# EPICS StreamDevice protocol: epics_installer_v1.0/option/serialTest_RAON_20220420/db/A100L.proto
ReplyTimeout = 500;
InTerminator = CR;

# No outTerminator because we need to send ENQ clean or RS485 will mess up the reply.

#address = ESC "0\$1"; # for RS485

set_onoff
{
    out "#\$1%{SYSOFF|SYSON}" CR;
    in  "#\$1 OK..";
}

read_status
{
    out "#\$1STA" CR;
    in "#\$1"
       " "
       "%(\$2:STATUS-PUMP_RUNNING)1d"
       "000000000"
       "%r"
       " 0000 0000 000 000 000 0000 00 000000"
       "%(\$2:FrequencyControlDefect)01d"
       "%02r"
       "%(\$2:MotorTemperatureDefect)01d"
       "%03r"
       "%(\$2:MaintenanceDefect)01d"
       "%012r";
}

set_address
{
    out "#\$1ADR%d" CR;
    in "#%d OK..";
}
